TYPE ST_LIST_CTRL :
STRUCT
  Cmd         : E_LIST_CTRL;
END_STRUCT
END_TYPE

(* stored: Version 1.1.0.1
   DUT ST_LIST_CTRL: Id {2a017b90-7695-44be-8d0a-cd24cc4baaca} *)
